{attribute 'GeneratedUsingTerminal: EL3783-0000-0018'}
{attribute addProperty BoxType "EL3783-0000-0018"}
{attribute addProperty Id "U3_SamplesAT %I*U3_Samples_1109DCAA40"}
{attribute addProperty CRC "2409861949"}
{attribute addProperty Size "40"}
TYPE L3_Voltage_Samples_8FA3933D EXTENDS InputBase_8311D824 :
STRUCT
	{attribute addProperty Name "U3_Samples"}
	U3_Samples AT %I* : U3_Samples_1109DCAA;
END_STRUCT
END_TYPE

(* stored: Version 1.2.0.0, ProductVersion 3.1.4024.11
   DUT L3_Voltage_Samples_8FA3933D: Id {f61db0fa-2178-419c-9fdd-b88ae72e9954} *)
